DATA_BLOCK "ServoV90_DeviceCtl"
VAR
  V90Servo : Array[1..4] of Struct;
END_VAR
BEGIN
END_DATA_BLOCK
